FUNCTION_BLOCK "FbBlink"
TITLE = Мигающий светодиод.
{ S7_Optimized_Access := 'FALSE' }
AUTHOR : VA
FAMILY : LIB_PLC
VERSION : 1.2
   VAR_INPUT
      TimeOn : DInt := L#2000;   // Время включения лампочки [мс].
      TimeOff : DInt := L#2000;   // Время выключения лампочки [мс].
      Ts_ms : DInt := L#100;   // Шаг дискретизации по времени [мс].
      Reset : Bool;   // Сброс при перезагрузке.
   END_VAR

   VAR_OUTPUT
      BlinkLamp : Bool;   // Мигающая лампочка.
   END_VAR

   VAR
      Timer1 : DInt;   // Таймер1 [мс].
      State1 : Int;   // Граф состояний.
   END_VAR

   VAR CONSTANT
      STATE_RESET : Int;
      STATE_ON : Int := 1;
      STATE_OFF : Int := 2;
   END_VAR


BEGIN


	// Мигающий светодиод.
	//            DbBlink
	//    +---------------------+
	//    |       FbBlink       |
	//   -|TimeOn      BlinkLamp|->-
	//   -|TimeOff              |
	//   -|Ts_ms                |
	//   -|Reset                |
	//    +---------------------+

	// Пример построения универсального кроссплатформенного графа состояний.
	// Использую этот код как заготовку под более сложные алгоритмы.
	// Данный алгоритм гораздо быстрее разрабатывать чем конечный автомат с памятью.

	IF (#Reset) THEN // Сброс при перезагрузке.
	#State1 := #STATE_RESET;
	END_IF;

	CASE (#State1) OF // Граф состояний.

	#STATE_RESET: // Сброс.
	#BlinkLamp := FALSE;
	#Timer1    := 0;
	#State1 := #STATE_ON;

	#STATE_ON: // Включить лампочку на заданное время.
	#BlinkLamp := TRUE;
	#Timer1 := #Timer1 + #Ts_ms;
	IF (#Timer1 >= #TimeOn) THEN
	#State1 := #STATE_OFF;
	#Timer1 := 0;
	END_IF;

	#STATE_OFF: // Выключить лампочку на заданное время.
	#BlinkLamp := FALSE;
	#Timer1 := #Timer1 + #Ts_ms;
	IF (#Timer1 >= #TimeOff) THEN
	#State1 := #STATE_ON;
	#Timer1 := 0;
	END_IF;

	ELSE // RESET при неопределенном состоянии.
	#State1 := #STATE_RESET;
	END_CASE; // CASE (State1) OF

	// Граф состояний.
	//
	//            |
	//           -+- Reset
	//            |
	//            V
	//  +-------------------+
	//  | State1 =          |
	//  | STATE_RESET       |
	//  | BlinkLamp = 0     |
	//  +-------------------+
	//            |
	//            |
	//            |
	//            |
	//            V
	//  +-------------------+
	//  | State1 =          |
	//  | STATE_ON          |<--------------+
	//  | BlinkLamp = 1     |               |
	//  +-------------------+               |
	//            |                         |
	//            |                         |
	//           -+- Timer1 >= TimeOn      -+- Timer1 >= TimeOff
	//            |                         |
	//            V                         |
	//  +-------------------+               |
	//  | State1 =          |               |
	//  | STATE_OFF         |---------------+
	//  | BlinkLamp = 0     |
	//  +-------------------+

	// @COPYLEFT ALL WRONGS RESERVED :)
	// Author: VA
	// Contacts: DIY.PLC.314@gmail.com
	// Date start LIB_PLC: 2014
	// License: GNU GPL-2.0-or-later
	// https://www.gnu.org/licenses/old-licenses/gpl-2.0.html
	// https://www.youtube.com/watch?v=n1F_MfLRlX0
	// https://www.youtube.com/@DIY_PLC
	// https://github.com/DIYPLC/LIB_PLC
	// https://oshwlab.com/diy.plc.314/PLC_HW1_SW1
	// https://3dtoday.ru/3d-models/mechanical-parts/body/korpus-na-din-reiku
	// https://t.me/DIY_PLC


END_FUNCTION_BLOCK

